// TIA Portal project "Project2" (V20)

(* hardware
DEVICE "S7-1500/ET200MP station_1"  S7-1500 station
   slot 0: "Rail_0"  Rack  6ES7 590-1***0-0AA0
   slot 1: "Brain"  CPU 1512C-1 PN  6ES7 512-1CK00-0AB0  V1.8
      slot 3: "CPU display_1"  6ES7591-1AA00-0AA0
      slot 32768: "PROFINET interface_1"  X1
         slot 32769: "Port_1"  X1 P1
         slot 32770: "Port_2"  X1 P2
   slot 2: "DI 16x24VDC / DQ 16x24VDC/0.5A BA_1"  DI 16x24VDC/DQ 16x24VDC/0.5A BA  6ES7 523-1BL00-0AA0  V1.1
*)

// ===== PLC "Brain"  CPU 1512C-1 PN =====

VAR_GLOBAL   // PLC tag table "Conveyor 1"
   "B1" AT %I10.0 : Bool;   // Component at Conveyor Start
   "B2" AT %I10.1 : Bool;   // Component at Conveyor Center
   "B3" AT %I10.2 : Bool;   // No Component at Conveyor End
   "S1" AT %I10.3 : Bool;   // Start Button
   "K1" AT %Q4.0 : Bool;   // Conveyor Belt On
   "1M1" AT %Q4.1 : Bool;   // Open Stopper
   "P1" AT %Q4.2 : Bool;   // Indicator LED
   "B20" AT %I10.4 : Bool;   // Color Detection
   "K1.1" AT %Q4.3 : Bool;   // Conveyor Belt Reverse
END_VAR

VAR_GLOBAL   // PLC tag table "Clock Memory"
   "Clock_Byte" AT %MB0 : Byte;
   "Clock_10Hz" AT %M0.0 : Bool;
   "Clock_5Hz" AT %M0.1 : Bool;
   "Clock_2.5Hz" AT %M0.2 : Bool;
   "Clock_2Hz" AT %M0.3 : Bool;
   "Clock_1.25Hz" AT %M0.4 : Bool;
   "Clock_1Hz" AT %M0.5 : Bool;
   "Clock_0.625Hz" AT %M0.6 : Bool;
   "Clock_0.5Hz" AT %M0.7 : Bool;
   "Stop Button" AT %I12.0 : Bool;
   "Reset Mode Selected" AT %I12.1 : Bool;
   "Automatic Mode Selected" AT %I12.2 : Bool;
   "Tap Mode Selected" AT %I12.3 : Bool;
   "Next Step Button" AT %I12.4 : Bool;
END_VAR

VAR_GLOBAL   // PLC tag table "Conveyor 2"
   "B4" AT %I11.0 : Bool;   // Component at Conveyor Start
   "B5" AT %I11.1 : Bool;   // Component at Conveyor Center
   "B6" AT %I11.2 : Bool;   // No Component at Conveyor End
   "K2" AT %Q5.0 : Bool;   // Conveyor Belt On
   "2M1" AT %Q5.1 : Bool;   // Open Stopper
   "P2" AT %Q5.2 : Bool;   // Indicator LED
END_VAR

DATA_BLOCK "Conveyor Sequence_DB"   // DB1
{ S7_Optimized_Access := 'TRUE' }
VERSION : 0.1
// stored: InstanceOfName Conveyor Sequence
"Conveyor Sequence"
BEGIN
END_DATA_BLOCK

FUNCTION_BLOCK "Conveyor Sequence"   // FB1, GRAPH_PLUS
{ S7_Optimized_Access := 'TRUE' }
VERSION : 0.1
   VAR_INPUT
      OFF_SQ : Bool := false;   // Turn sequence off
      INIT_SQ : Bool := false;   // Set sequence to initial state
      ACK_EF : Bool := false;   // Acknowledge all errors and faults
      S_PREV : Bool := false;   // Output previous step in parameter S_NO
      S_NEXT : Bool := false;   // Indicate next step in parameter S_NO
      SW_AUTO : Bool := false;   // Automatic mode
      SW_TAP : Bool := false;   // Semiautomatic/switch with transition
      SW_TOP : Bool := false;   // Semiautomatic/ignore transition
      SW_MAN : Bool := false;   // Manual mode
      S_SEL : Int := 0;   // Select step to be output to S_NO
      S_ON : Bool := false;   // Activate step indicated in S_NO
      S_OFF : Bool := false;   // Disable step indicated in S_NO
      T_PUSH : Bool := false;   // Enable transition to switch in semi automatic mode
   END_VAR
   VAR_OUTPUT
      S_NO : Int := 0;   // Step number
      S_MORE : Bool := false;   // More steps are available and can be shown in S_NO
      S_ACTIVE : Bool := false;   // Step indicated in S_NO is active
      ERR_FLT : Bool := false;   // Interlock or supervision group error
      AUTO_ON : Bool := false;   // Automatic mode is active
      TAP_ON : Bool := false;   // Semiautomatic mode/step with transition enabled
      TOP_ON : Bool := false;   // Semiautomatic mode/ignore transition enabled
      MAN_ON : Bool := false;   // Manual mode is active
   END_VAR
   VAR
      HMI_INFO : Array[0..8] of UInt;
      IF_PAR : G7_IfParPlus_V2;
      RT_DATA : G7_RTDataPlus_V2;   // Internal data area
      "Waiting for Piece" : G7_TransitionPlus_V2;   // Transition structure
      "In Center Position" : G7_TransitionPlus_V2;   // Transition structure
      "Not in Center Position" : G7_TransitionPlus_V2;   // Transition structure
      "In End Position" : G7_TransitionPlus_V2;   // Transition structure
      "Belt Empty" : G7_TransitionPlus_V2;   // Transition structure
      "Initial Step" : G7_StepPlus_V2;   // Step structure
      "Start Conveyor" : G7_StepPlus_V2;   // Step structure
      "Open Stopper" : G7_StepPlus_V2;   // Step structure
      "Continue Conveyor" : G7_StepPlus_V2;   // Step structure
      "Wait for empty  belt" : G7_StepPlus_V2;   // Step structure
      SINI : Array[0..1] of USInt;
      LSTT : Array[0..4] of USInt;
      ATAJ : Array[0..4] of USInt;
      ATAB : Array[0..4] of USInt;
      PSTT : Array[0..4] of USInt;
      NSTT : Array[0..4] of USInt;
      ASSJ : Array[0..4] of USInt;
      ASSB : Array[0..4] of USInt;
      PTTS : Array[0..4] of USInt;
      NTTS : Array[0..4] of USInt;
      SW_SQTS : Array[0..4] of USInt;
      SWITCH : Array[0..0] of USInt;
      TVX : Array[0..1] of USInt;
      TTX : Array[0..1] of USInt;
      TSX : Array[0..1] of USInt;
      S00X : Array[0..1] of USInt;
      SOFFX : Array[0..1] of USInt;
      SONX : Array[0..1] of USInt;
      SAX : Array[0..1] of USInt;
      SERRX : Array[0..5] of USInt;
      SMX : Array[0..5] of USInt;
      S0X : Array[0..5] of USInt;
      S1X : Array[0..5] of USInt;
      IL_ALARM_INST : Program_Alarm;
      SUP_ALARM_INST : Program_Alarm;
      STEP_TIME_ALARM_INST : Program_Alarm;
      IEC_TIMER_INST : IEC_TIMER;
      TRANSACTION_FLAG : Bool := false;
      "Grey Part In Center" : G7_TransitionPlus_V2;   // Transition structure
      "Conveyor Reverse" : G7_StepPlus_V2;   // Step structure
      "Back at Start" : G7_TransitionPlus_V2;   // Transition structure
      "Wait for Empty" : G7_StepPlus_V2;   // Step structure
      Trans8 : G7_TransitionPlus_V2;   // Transition structure
   END_VAR
   // SINI[0] := 2;
   // LSTT[0] := 255;
   // LSTT[1] := 255;
   // LSTT[2] := 255;
   // LSTT[3] := 255;
   // ATAJ[1] := 1;
   // ATAJ[2] := 2;
   // ATAJ[3] := 3;
   // ATAJ[4] := 4;
   // ATAB[1] := 1;
   // ATAB[2] := 2;
   // ATAB[3] := 3;
   // ATAB[4] := 4;
   // PSTT[1] := 1;
   // PSTT[2] := 2;
   // PSTT[3] := 3;
   // PSTT[4] := 4;
   // NSTT[0] := 1;
   // NSTT[1] := 2;
   // NSTT[2] := 3;
   // NSTT[3] := 4;
   // ASSJ[1] := 1;
   // ASSJ[2] := 2;
   // ASSJ[3] := 3;
   // ASSJ[4] := 4;
   // ASSB[1] := 1;
   // ASSB[2] := 2;
   // ASSB[3] := 3;
   // ASSB[4] := 4;
   // PTTS[0] := 255;
   // PTTS[2] := 1;
   // PTTS[3] := 2;
   // PTTS[4] := 3;
   // NTTS[1] := 1;
   // NTTS[2] := 2;
   // NTTS[3] := 3;
   // NTTS[4] := 4;
   // TVX[0] := 16#1;
   // TTX[0] := 16#1;
   // TSX[0] := 16#1;
   // S00X[0] := 16#1;
   // SOFFX[0] := 16#1;
   // SONX[0] := 16#1;
   // SAX[0] := 16#1;
   // SERRX[0] := 16#1;
   // SMX[0] := 16#1;
   // S0X[0] := 16#1;
   // S1X[0] := 16#1;
BEGIN
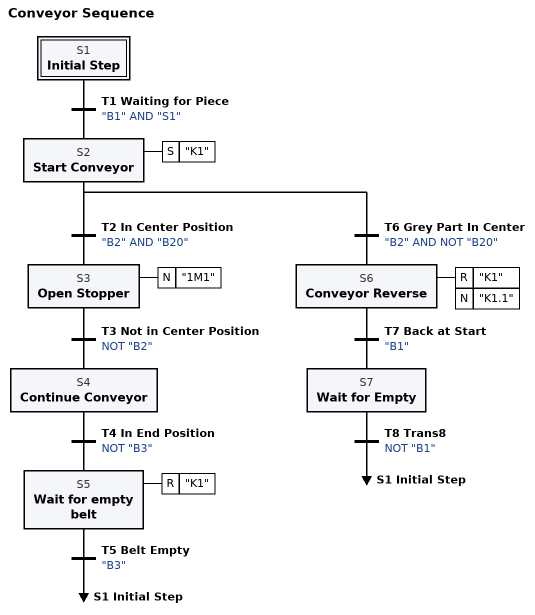
   // sequencer 1
   INITIAL_STEP "Initial Step":   // S1, max time T#10S, warning time T#7S
   END_STEP
   TRANSITION "Waiting for Piece" FROM "Initial Step" TO "Start Conveyor"   // T1
      := "B1" AND "S1";
   END_TRANSITION
   STEP "Start Conveyor":   // S2, max time T#10S, warning time T#7S
              S    "K1"
   END_STEP
   TRANSITION "In Center Position" FROM "Start Conveyor" TO "Open Stopper"   // T2
      := "B2" AND "B20";
   END_TRANSITION
   TRANSITION "Grey Part In Center" FROM "Start Conveyor" TO "Conveyor Reverse"   // T6
      := "B2" AND NOT "B20";
   END_TRANSITION
   STEP "Open Stopper":   // S3, max time T#10S, warning time T#7S
              N    "1M1"
   END_STEP
   TRANSITION "Not in Center Position" FROM "Open Stopper" TO "Continue Conveyor"   // T3
      := NOT "B2";
   END_TRANSITION
   STEP "Continue Conveyor":   // S4, max time T#10S, warning time T#7S
   END_STEP
   TRANSITION "In End Position" FROM "Continue Conveyor" TO "Wait for empty  belt"   // T4
      := NOT "B3";
   END_TRANSITION
   STEP "Wait for empty  belt":   // S5, max time T#10S, warning time T#7S
              R    "K1"
   END_STEP
   TRANSITION "Belt Empty" FROM "Wait for empty  belt" TO "Initial Step"   // T5, jump
      := "B3";
   END_TRANSITION
   STEP "Conveyor Reverse":   // S6, max time T#10S, warning time T#7S
              R    "K1"
              N    "K1.1"
   END_STEP
   TRANSITION "Back at Start" FROM "Conveyor Reverse" TO "Wait for Empty"   // T7
      := "B1";
   END_TRANSITION
   STEP "Wait for Empty":   // S7, max time T#10S, warning time T#7S
   END_STEP
   TRANSITION Trans8 FROM "Wait for Empty" TO "Initial Step"   // T8, jump
      := NOT "B1";
   END_TRANSITION
END_FUNCTION_BLOCK

FUNCTION "Conveyor" : Void   // FC1, LAD
{ S7_Optimized_Access := 'TRUE' }
VERSION : 0.1
   VAR_INPUT
      "Conveyor Start" : Bool;
      "Conveyor Center" : Bool;
      "Conveyor End" : Bool;
      "Start Button" : Bool;
      "Conveyor On Frequency" : Bool;
      "Part at Start Frequency" : Bool;
   END_VAR
   VAR_OUTPUT
      Stopper : Bool;
      LED : Bool;
   END_VAR
   VAR_IN_OUT
      Conveyor : Bool;
   END_VAR
BEGIN

REGION Network 1
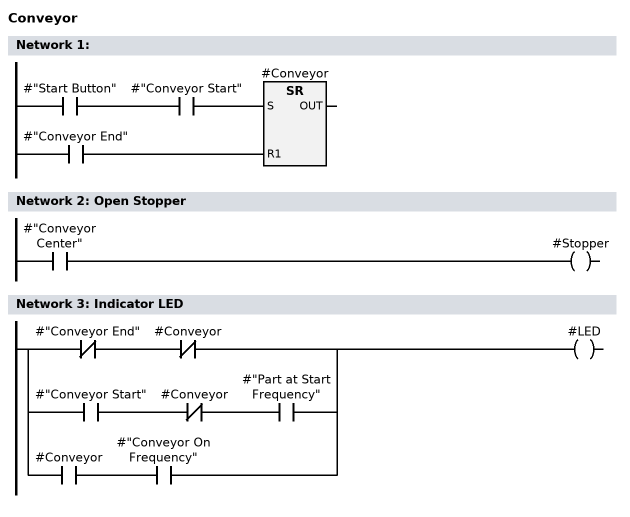
   RUNG wire#powerrail
      Contact( #"Start Button" )
      Contact( #"Conveyor Start" )
      S_SR(operand := #Conveyor, r1 := wire#w1)
   END_RUNG
   RUNG wire#powerrail
      Contact( #"Conveyor End" )
   END_RUNG wire#w1
   // the same network as SCL:
   IF #"Start Button" AND #"Conveyor Start" THEN
       #Conveyor := TRUE;   // SR flip-flop
   END_IF;
   IF #"Conveyor End" THEN #Conveyor := FALSE; END_IF;
END_REGION

REGION Network 2: Open Stopper
   RUNG wire#powerrail
      Contact( #"Conveyor Center" )
      Coil( #Stopper )
   END_RUNG
   // the same network as SCL:
   #Stopper := #"Conveyor Center";
END_REGION

REGION Network 3: Indicator LED
   RUNG wire#powerrail
      I_Contact( #"Conveyor End" )
      I_Contact( #Conveyor )
      wire#w1
      Coil( #LED )
   END_RUNG
   RUNG wire#powerrail
      Contact( #"Conveyor Start" )
      I_Contact( #Conveyor )
      Contact( #"Part at Start Frequency" )
   END_RUNG wire#w1
   RUNG wire#powerrail
      Contact( #Conveyor )
      Contact( #"Conveyor On Frequency" )
   END_RUNG wire#w1
   // the same network as SCL:
   #LED := (NOT #"Conveyor End" AND NOT #Conveyor) OR (#"Conveyor Start" AND NOT #Conveyor AND #"Part at Start Frequency") OR (#Conveyor AND #"Conveyor On Frequency");
END_REGION
END_FUNCTION

ORGANIZATION_BLOCK "Main"   // OB1, LAD, ProgramCycle
TITLE = "Main Program Sweep (Cycle)"
{ S7_Optimized_Access := 'TRUE' }
VERSION : 0.1
   VAR_INPUT
      Initial_Call : Bool;   // Initial call of this OB
      Remanence : Bool;   // =True, if remanent data are available
   END_VAR
BEGIN

REGION Network 1
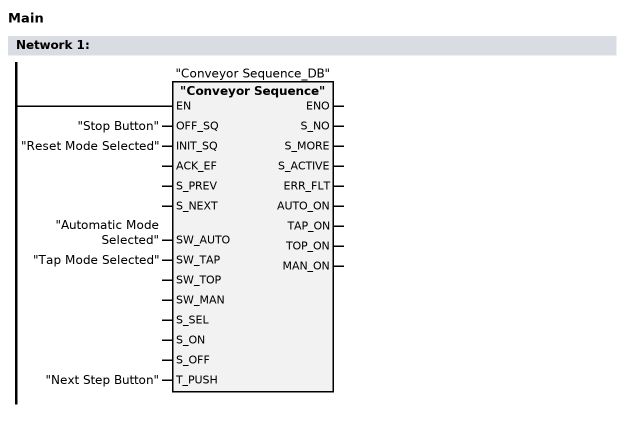
   RUNG wire#powerrail
      "Conveyor Sequence_DB"(OFF_SQ := "Stop Button", INIT_SQ := "Reset Mode Selected", ACK_EF :=, S_PREV :=, S_NEXT :=, SW_AUTO := "Automatic Mode Selected", SW_TAP := "Tap Mode Selected", SW_TOP :=, SW_MAN :=, S_SEL :=, S_ON :=, S_OFF :=, T_PUSH := "Next Step Button", S_NO =>, S_MORE =>, S_ACTIVE =>, ERR_FLT =>, AUTO_ON =>, TAP_ON =>, TOP_ON =>, MAN_ON =>)
   END_RUNG
   // the same network as SCL:
   "Conveyor Sequence_DB"(OFF_SQ := "Stop Button",   // "Conveyor Sequence"
                          INIT_SQ := "Reset Mode Selected",
                          SW_AUTO := "Automatic Mode Selected",
                          SW_TAP := "Tap Mode Selected",
                          T_PUSH := "Next Step Button");
END_REGION
END_ORGANIZATION_BLOCK